TYPE (* IEC61131-3, Table 14#5 *)
  (* Standard: 1131-3 *)
  (* Version 0.0, 1/8/2024, Cheyan, Schneider Electric, Template *)
  PACKAGE Main;
  {SET_ATTRIBUTE(nxtDataType, 9gA4evvp0K3sYuYBrz+XyN166j18T5K4IShRdiIPcNBe4lxG1OllktWrZu5DnBj5bF0C1aNk6OBPmbiKVFxsH7CikOATqeigb8G7rpytc65C4Su2Rxwz5kb43Yb/BKy0)}
  SPS : STRUCT
    stVal : BOOL;
    q : Quality;
    t : TimeStamp;
  END_STRUCT;
END_TYPE
